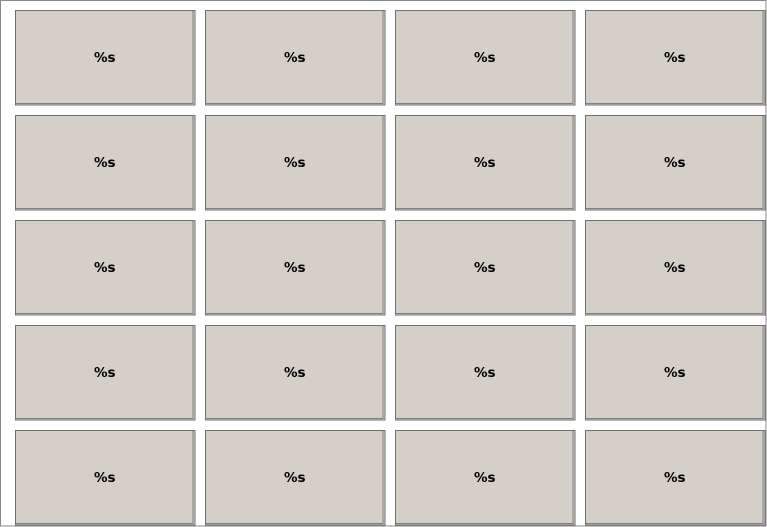
VISUALIZATION VISU_AxesManual_Positions  // 767x527
VAR_IN_OUT
	ref : Axes;
    widget : AxesManualPositionsWidget;
END_VAR
    Button (15,10 180x95), "%s", text variable: ref.config.knownPositions.position0.name, invisible if: widget.invisiblePosition0, input disabled if: ref.processes.moveKnownPosition.statuses.enabledStatus.disabled
        OnMouseClick: execute { ref.processes.moveKnownPosition.request(ref.config.knownPositions.position0.name); }
    Button (15,115 180x95), "%s", text variable: ref.config.knownPositions.position1.name, invisible if: widget.invisiblePosition1, input disabled if: ref.processes.moveKnownPosition.statuses.enabledStatus.disabled
        OnMouseClick: execute { ref.processes.moveKnownPosition.request(ref.config.knownPositions.position1.name); }
    Button (15,220 180x95), "%s", text variable: ref.config.knownPositions.position2.name, invisible if: widget.invisiblePosition2, input disabled if: ref.processes.moveKnownPosition.statuses.enabledStatus.disabled
        OnMouseClick: execute { ref.processes.moveKnownPosition.request(ref.config.knownPositions.position2.name); }
    Button (15,325 180x95), "%s", text variable: ref.config.knownPositions.position3.name, invisible if: widget.invisiblePosition3, input disabled if: ref.processes.moveKnownPosition.statuses.enabledStatus.disabled
        OnMouseClick: execute { ref.processes.moveKnownPosition.request(ref.config.knownPositions.position3.name); }
    Button (15,430 180x95), "%s", text variable: ref.config.knownPositions.position4.name, invisible if: widget.invisiblePosition4, input disabled if: ref.processes.moveKnownPosition.statuses.enabledStatus.disabled
        OnMouseClick: execute { ref.processes.moveKnownPosition.request(ref.config.knownPositions.position4.name); }
    Button (205,10 180x95), "%s", text variable: ref.config.knownPositions.position5.name, invisible if: widget.invisiblePosition5, input disabled if: ref.processes.moveKnownPosition.statuses.enabledStatus.disabled
        OnMouseClick: execute { ref.processes.moveKnownPosition.request(ref.config.knownPositions.position5.name); }
    Button (205,115 180x95), "%s", text variable: ref.config.knownPositions.position6.name, invisible if: widget.invisiblePosition6, input disabled if: ref.processes.moveKnownPosition.statuses.enabledStatus.disabled
        OnMouseClick: execute { ref.processes.moveKnownPosition.request(ref.config.knownPositions.position6.name); }
    Button (205,220 180x95), "%s", text variable: ref.config.knownPositions.position7.name, invisible if: widget.invisiblePosition7, input disabled if: ref.processes.moveKnownPosition.statuses.enabledStatus.disabled
        OnMouseClick: execute { ref.processes.moveKnownPosition.request(ref.config.knownPositions.position7.name); }
    Button (205,325 180x95), "%s", text variable: ref.config.knownPositions.position8.name, invisible if: widget.invisiblePosition8, input disabled if: ref.processes.moveKnownPosition.statuses.enabledStatus.disabled
        OnMouseClick: execute { ref.processes.moveKnownPosition.request(ref.config.knownPositions.position8.name); }
    Button (205,430 180x95), "%s", text variable: ref.config.knownPositions.position9.name, invisible if: widget.invisiblePosition9, input disabled if: ref.processes.moveKnownPosition.statuses.enabledStatus.disabled
        OnMouseClick: execute { ref.processes.moveKnownPosition.request(ref.config.knownPositions.position9.name); }
    Button (395,10 180x95), "%s", text variable: ref.config.knownPositions.position10.name, invisible if: widget.invisiblePosition10, input disabled if: ref.processes.moveKnownPosition.statuses.enabledStatus.disabled
        OnMouseClick: execute { ref.processes.moveKnownPosition.request(ref.config.knownPositions.position10.name); }
    Button (395,115 180x95), "%s", text variable: ref.config.knownPositions.position11.name, invisible if: widget.invisiblePosition11, input disabled if: ref.processes.moveKnownPosition.statuses.enabledStatus.disabled
        OnMouseClick: execute { ref.processes.moveKnownPosition.request(ref.config.knownPositions.position11.name); }
    Button (395,220 180x95), "%s", text variable: ref.config.knownPositions.position12.name, invisible if: widget.invisiblePosition12, input disabled if: ref.processes.moveKnownPosition.statuses.enabledStatus.disabled
        OnMouseClick: execute { ref.processes.moveKnownPosition.request(ref.config.knownPositions.position12.name); }
    Button (395,325 180x95), "%s", text variable: ref.config.knownPositions.position13.name, invisible if: widget.invisiblePosition13, input disabled if: ref.processes.moveKnownPosition.statuses.enabledStatus.disabled
        OnMouseClick: execute { ref.processes.moveKnownPosition.request(ref.config.knownPositions.position13.name); }
    Button (395,430 180x95), "%s", text variable: ref.config.knownPositions.position14.name, invisible if: widget.invisiblePosition14, input disabled if: ref.processes.moveKnownPosition.statuses.enabledStatus.disabled
        OnMouseClick: execute { ref.processes.moveKnownPosition.request(ref.config.knownPositions.position14.name); }
    Button (585,10 180x95), "%s", text variable: ref.config.knownPositions.position15.name, invisible if: widget.invisiblePosition15, input disabled if: ref.processes.moveKnownPosition.statuses.enabledStatus.disabled
        OnMouseClick: execute { ref.processes.moveKnownPosition.request(ref.config.knownPositions.position15.name); }
    Button (585,115 180x95), "%s", text variable: ref.config.knownPositions.position16.name, invisible if: widget.invisiblePosition16, input disabled if: ref.processes.moveKnownPosition.statuses.enabledStatus.disabled
        OnMouseClick: execute { ref.processes.moveKnownPosition.request(ref.config.knownPositions.position16.name); }
    Button (585,220 180x95), "%s", text variable: ref.config.knownPositions.position17.name, invisible if: widget.invisiblePosition17, input disabled if: ref.processes.moveKnownPosition.statuses.enabledStatus.disabled
        OnMouseClick: execute { ref.processes.moveKnownPosition.request(ref.config.knownPositions.position17.name); }
    Button (585,325 180x95), "%s", text variable: ref.config.knownPositions.position18.name, invisible if: widget.invisiblePosition18, input disabled if: ref.processes.moveKnownPosition.statuses.enabledStatus.disabled
        OnMouseClick: execute { ref.processes.moveKnownPosition.request(ref.config.knownPositions.position18.name); }
    Button (585,430 180x95), "%s", text variable: ref.config.knownPositions.position19.name, invisible if: widget.invisiblePosition19, input disabled if: ref.processes.moveKnownPosition.statuses.enabledStatus.disabled
        OnMouseClick: execute { ref.processes.moveKnownPosition.request(ref.config.knownPositions.position19.name); }
END_VISUALIZATION

(* stored: Version 1.1.0.1, ProductVersion 3.1.4019.2
   Visu VISU_AxesManual_Positions: Id {fc727c57-51bb-4dc4-85f2-c00b55e1f4ea} *)
